# B&R Automation Studio project DuctLines (part 4)

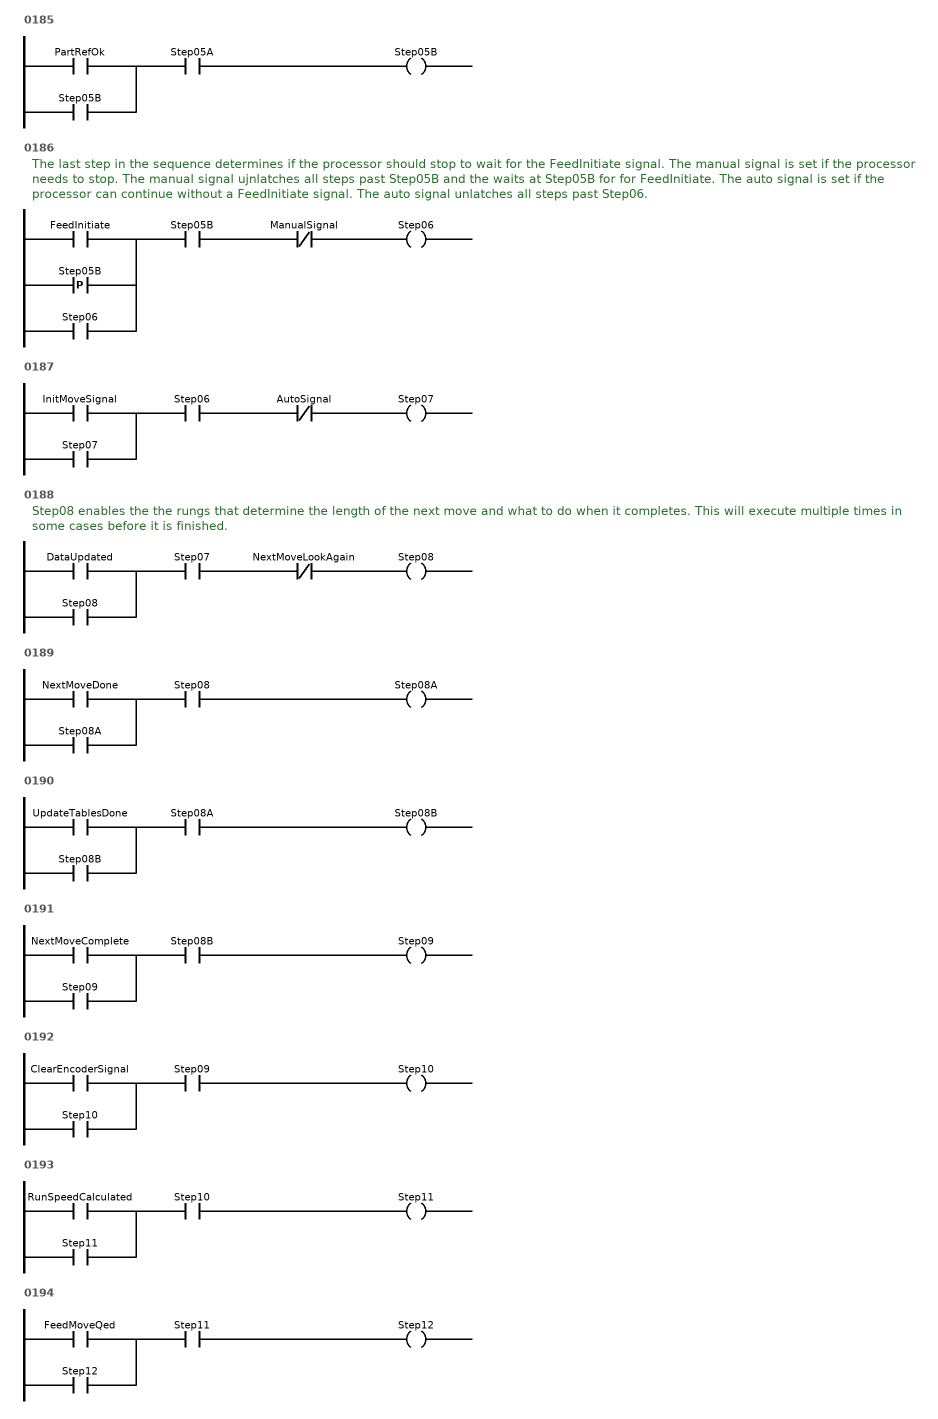
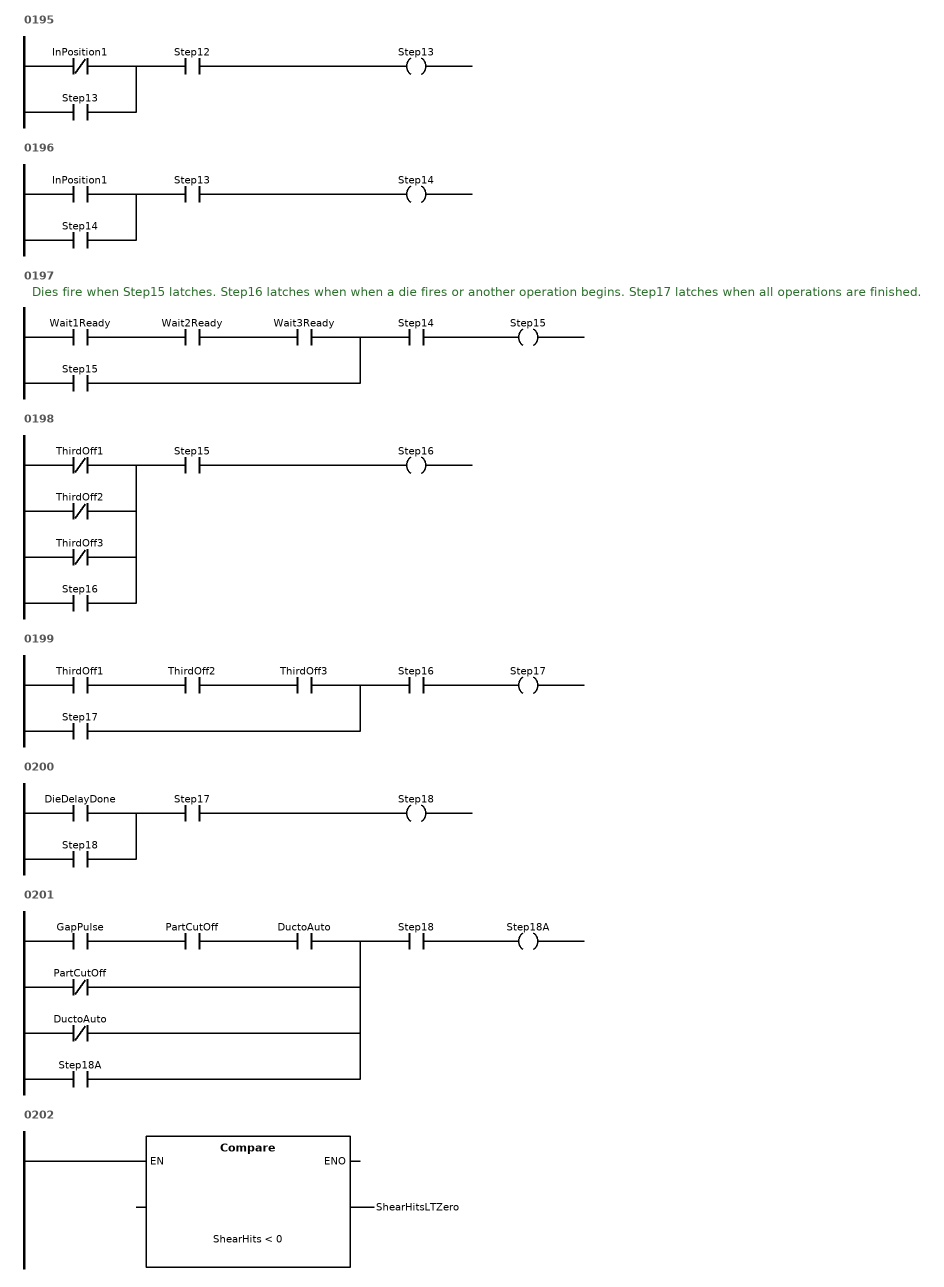
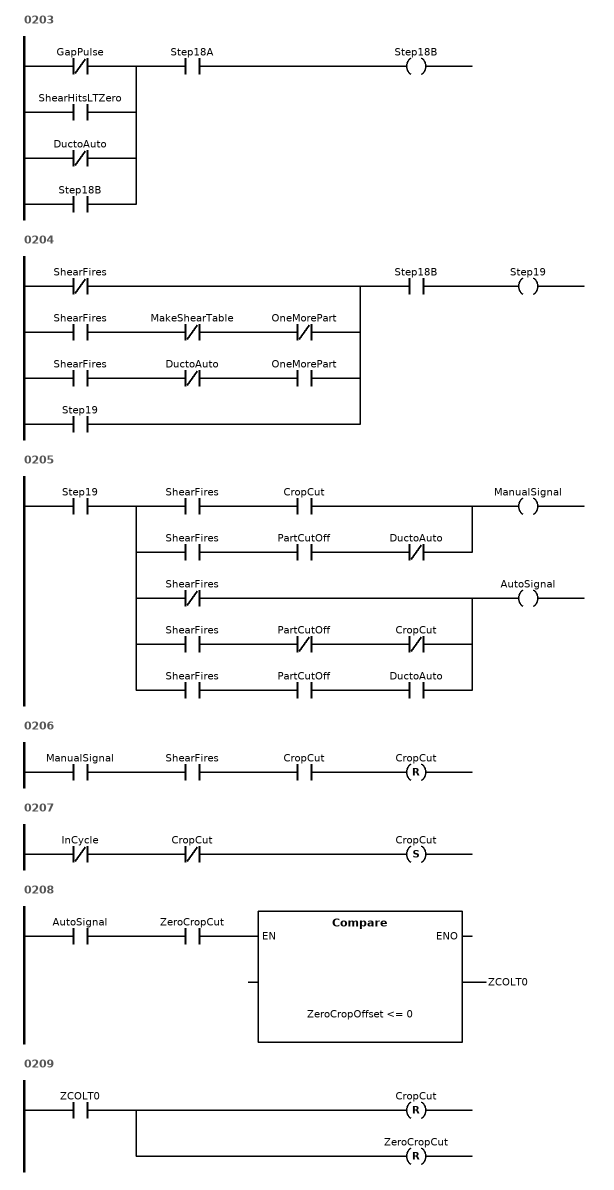
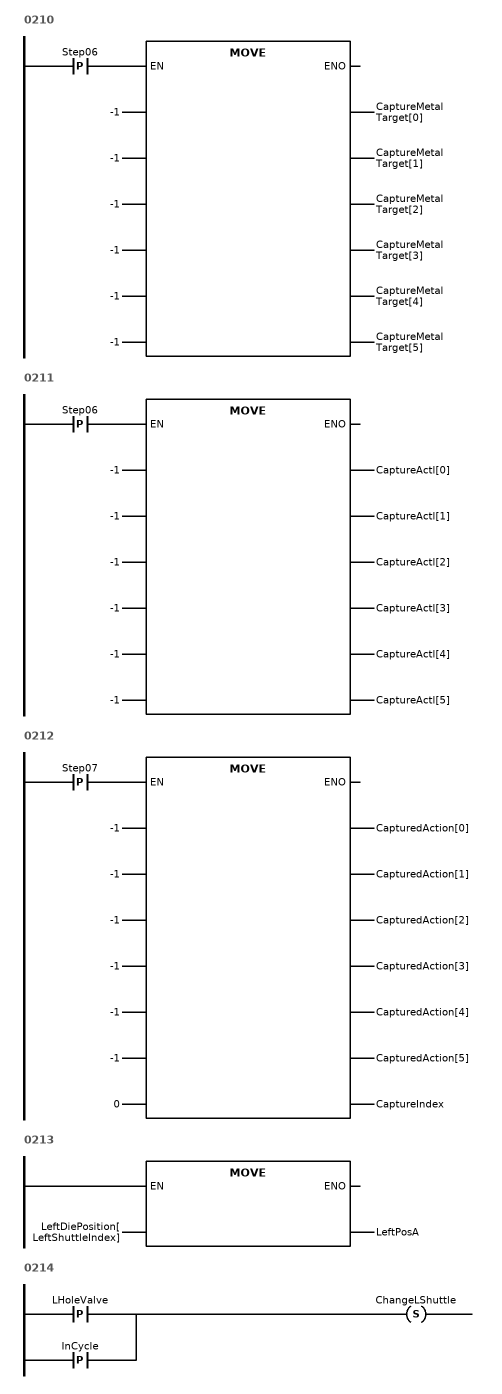
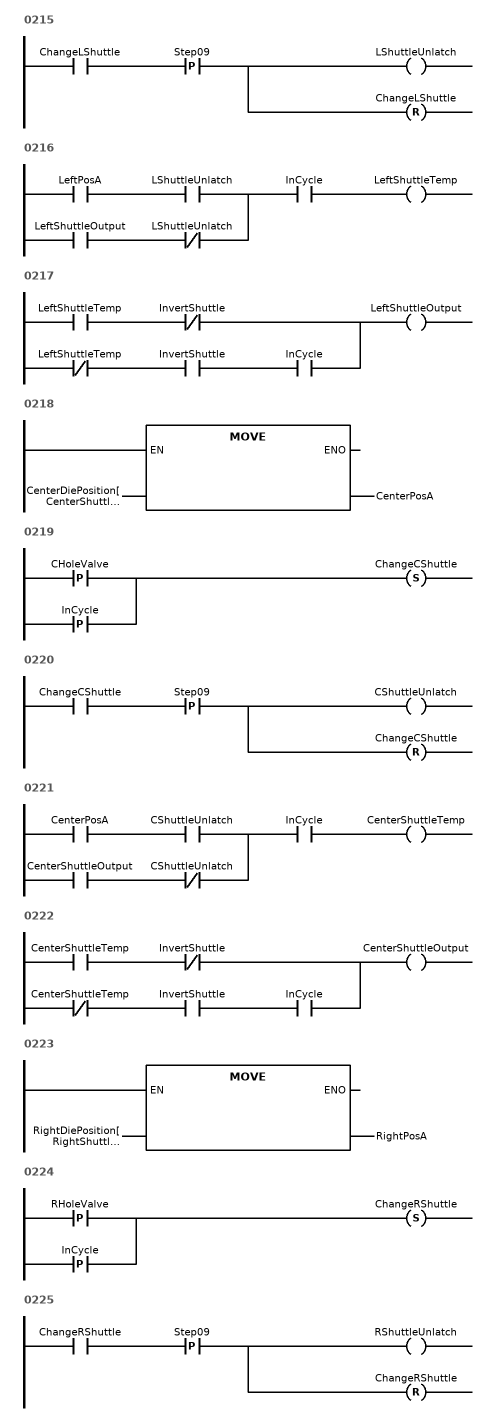
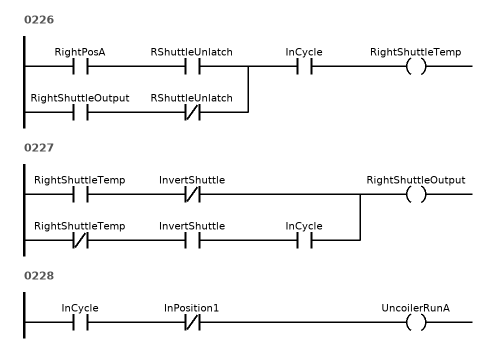
Ladder, written as Structured Text:
```iecst
PROGRAM _CYCLIC
VAR
    _e1 : R_TRIG;
    _e2 : R_TRIG;
    _e3 : F_TRIG;
    _e4 : F_TRIG;
    _e5 : R_TRIG;
    _e6 : F_TRIG;
    _e7 : F_TRIG;
    _e8 : F_TRIG;
    _e9 : R_TRIG;
    _p10 : BOOL;
    _e11 : R_TRIG;
    _e12 : R_TRIG;
    _e13 : R_TRIG;
    _e14 : F_TRIG;
    _e15 : F_TRIG;
    _e16 : R_TRIG;
    _e17 : R_TRIG;
    _e18 : R_TRIG;
    _e19 : R_TRIG;
    _e20 : R_TRIG;
    _e21 : R_TRIG;
    _e22 : R_TRIG;
    _e23 : R_TRIG;
    _e24 : R_TRIG;
    _e25 : R_TRIG;
    _e26 : R_TRIG;
    _e27 : R_TRIG;
    _e28 : F_TRIG;
    _e29 : R_TRIG;
    _e30 : R_TRIG;
    _e31 : F_TRIG;
    _e32 : R_TRIG;
    _e33 : R_TRIG;
    _e34 : R_TRIG;
    _e35 : R_TRIG;
    _e36 : F_TRIG;
    _e37 : R_TRIG;
    _e38 : F_TRIG;
    _e39 : R_TRIG;
    _e40 : F_TRIG;
    _e41 : R_TRIG;
    _e42 : F_TRIG;
    _e43 : R_TRIG;
    _e44 : F_TRIG;
    _e45 : R_TRIG;
    _e46 : F_TRIG;
    _e47 : R_TRIG;
    _e48 : F_TRIG;
    _e49 : R_TRIG;
    _e50 : F_TRIG;
    _e51 : R_TRIG;
    _e52 : F_TRIG;
    _e53 : R_TRIG;
    _e54 : F_TRIG;
    _e55 : R_TRIG;
    _e56 : F_TRIG;
    _e57 : R_TRIG;
    _e58 : R_TRIG;
    _e59 : R_TRIG;
    _e60 : R_TRIG;
    _e61 : R_TRIG;
    _e62 : R_TRIG;
    _e63 : R_TRIG;
    _e64 : R_TRIG;
    _e65 : R_TRIG;
    _e66 : R_TRIG;
    _e67 : R_TRIG;
    _e68 : R_TRIG;
    _e69 : R_TRIG;
    _e70 : R_TRIG;
    _e71 : R_TRIG;
    _e72 : R_TRIG;
    _e73 : R_TRIG;
    _e74 : R_TRIG;
    _e75 : F_TRIG;
    _e76 : R_TRIG;
    _e77 : R_TRIG;
    _e78 : R_TRIG;
    _e79 : R_TRIG;
    _e80 : R_TRIG;
    _e81 : R_TRIG;
    _e82 : R_TRIG;
    _e83 : F_TRIG;
    _e84 : R_TRIG;
    _e85 : R_TRIG;
    _e86 : R_TRIG;
    _e87 : R_TRIG;
    _e88 : R_TRIG;
    _e89 : R_TRIG;
    _p90 : BOOL;
    _e91 : F_TRIG;
    _e92 : R_TRIG;
    _e93 : R_TRIG;
    _e94 : R_TRIG;
    _e95 : R_TRIG;
    _e96 : R_TRIG;
    _e97 : R_TRIG;
    _e98 : R_TRIG;
    _e99 : R_TRIG;
    _e100 : R_TRIG;
    _e101 : R_TRIG;
    _e102 : R_TRIG;
    _e103 : R_TRIG;
    _e104 : R_TRIG;
    _e105 : R_TRIG;
END_VAR
(* Network 1 *)
MetalEncoder := ActlMetalEncoder - CoilAccumulator;

(* Network 2 *)
AmberLight := ProcessorDriveEnable;

(* Network 3 *)
Analog1Forward := (ProcessorDriveEnable AND ProcessorJogFwd AND NOT InCycle) OR (Step04C AND NOT Step04D);

(* Network 4 *)
Analog1Reverse := (ProcessorDriveEnable AND ProcessorJogRev AND NOT InCycle) OR (Step04 AND NOT Step04B);

(* Network 5 *)
_e1(CLK := Analog1Forward);
IF _e1.Q THEN MotionStatus1 := 4; END_IF;

(* Network 6 *)
_e2(CLK := Analog1Reverse);
IF _e2.Q THEN MotionStatus1 := 5; END_IF;

(* Network 7 *)
_e3(CLK := Analog1Forward);
_e4(CLK := Analog1Reverse);
IF (_e3.Q OR _e4.Q) AND NOT StopFlag1 THEN StopFlag1 := TRUE; END_IF;

(* Network 8: ElectricDriveEnable Output *)
ElectricDriveEnable := MotionStatus1 >= 0;

(* Network 9: Blocking Valve Output *)
BlockingValve := ElectricDriveEnable OR ForceBlockingValve;

(* Network 10 *)
_e5(CLK := Step04E);
IF _e5.Q THEN MotionStatus1 := 0; END_IF;

(* Network 11 *)
_e6(CLK := InCycle);
IF _e6.Q THEN MotionStatus1 := -1; END_IF;

(* Network 12 *)
_e7(CLK := ProcessorDriveEnable);
IF _e7.Q THEN MotionStatus1 := -1; END_IF;

(* Network 13 *)
ServoLoop1Closed := (MotionStatus1 >= 0) AND (MotionStatus1 <= 3);

(* Network 14 *)
_e8(CLK := HumpLimitSwitch);
IF _e8.Q AND ServoLoop1Closed THEN MotionStatus1 := -1; END_IF;

(* Network 15: OneMorePart logic needs To Execute Before The FeedInitiate Signal rung. *)
JobChanging := (RunJob - 1)  <> ShearJob;

(* Network 16 *)
OneMorePart := (InCycle OR (OneMorePart AND NOT FeedInitiate)) AND JobChanging AND NOT RunContinuousSignal;

(* Network 17: Feed Initiate Signal *)
_e9(CLK := FeedInitButton);
_p10 := _e9.Q AND ProcessorDriveEnable AND MatlAtMeasureRoll;
FeedInitiate := _p10 AND (NOT ShearBrakeInstalled OR ShearBrakeReady);

(* Network 18: Verify HMI Job change request *)
IF RunJobClick AND NOT InCycle THEN NewRunJobOk := NewRunJob <= MaxRunJob; END_IF;

(* Network 19 *)
IF RunJobClick AND NewRunJobOk AND NOT InCycle THEN RunJob := NewRunJob; END_IF;

(* Network 20 *)
IF RunJobClick THEN NewRunJobOk := FALSE; END_IF;

(* Network 21 *)
IF RunJobClick THEN RunJobClick := FALSE; END_IF;

(* Network 22: Update HMI job when the shear finishes one. *)
JobsDifferent := (RunJob - 1) <> ShearJob;

(* Network 23 *)
ChangeJob1 := InCycle AND Step19 AND ShearFires AND JobsDifferent;

(* Network 24 *)
IF ChangeJob1 THEN RunJob := ShearJob + 1; END_IF;

(* Network 25 *)
_e11(CLK := FeedInitiate);
IF _e11.Q THEN NoShearHits := FALSE; END_IF;

(* Network 26: Latch BatchActive in whenever the FeedInitiate signal comes on and the Ducto Sequence isn't started. Step04 latches after PC downloads tables and resets StartSignal. Unlatch BatchActive at that point if the shear has no hits. Step19 is the last one in the Ducto sequence. If there are no shear hits, the run is finished. BatchActive unlatches and the entire sequence unlatches. *)
_e12(CLK := Step04);
IF Step19 OR _e12.Q THEN NoShearHits := ShearHits < 0; END_IF;

(* Network 27 *)
_e13(CLK := WarningComplete);
_e14(CLK := HumpLimitSwitch);
_e15(CLK := MatlAtMeasureRoll);
BatchCancelUnlatch := BatchCancelSignal OR NoShearHits OR NOT ProcessorDriveEnable OR (_e13.Q AND NOT FeedInitButton) OR _e14.Q OR _e15.Q;

(* Network 28 *)
InCycle := ((FeedInitiate AND NOT Step01) OR InCycle) AND NOT BatchCancelUnlatch;

(* Network 29 *)
BlueLight := InCycle;

(* Network 30: Turn Off The BatchActivePhysical Output momentarily To Unlatch The Physical Auto Circuit *)
Block_1 := (Step18 AND OneMorePart) OR (Block_1 AND DuctoAuto);

(* Network 31 *)
BatchActivePhysical := InCycle AND NOT Block_1;

(* Network 32: There are 3 of these timers *)
ZRCTon(IN := Step04A AND NOT Step04B, PT := T#500ms);
ZCReverseComplete := ZRCTon.Q;

(* Network 33 *)
DDDoneTimer(IN := Step04B AND NOT Step04C, PT := T#2s);
DirectionDelayDone := DDDoneTimer.Q;

(* Network 34 *)
ZCSCTimer(IN := Step04D, PT := T#2s);
ZCSettleComplete := ZCSCTimer.Q;

(* Network 35 *)
_e16(CLK := MatlAtMeasureRoll);
IF _e16.Q AND Step04C AND NOT Step04D THEN MetalEncoderLatch := ActlMetalEncoder; END_IF;

(* Network 36 *)
_e17(CLK := Step05A);
IF _e17.Q AND NOT ZeroCropCut THEN MetalEncoderLatch := ActlMetalEncoder; END_IF;

(* Network 37: First actions in Ducto sequence, reset indexes and moves, set start signal for PC to generate die tables. *)
IF Step01 AND NOT Step02 THEN
    ShearMove := 0.0;
    LTNotchMove := 0.0;
    VNotchMove := 0.0;
    LeftHoleMove := 0.0;
    CenterHoleMove := 0.0;
    RightHoleMove := 0.0;
    PartsMade := 0;
    ShearIndex := 0;
    LTNotchIndex := 0;
    VNotchIndex := 0;
    LeftHoleIndex := 0;
    CenterHoleIndex := 0;
    RightHoleIndex := 0;
    ButtonMove := 0.0;
    ShearBrakeMove := 0.0;
    CustomLTMove := 0.0;
    CleatMove := 0.0;
    ButtonIndex := 0;
    ShearBrakeIndex := 0;
    CustomLTIndex := 0;
END_IF;

(* Network 38 *)
IF Step01 AND NOT Step02 THEN
    CleatIndex := 0;
    ButtonActual := 0;
    CustomVMove := 0.0;
    CustomVIndex := 0;
    BeadRollMove := 0.0;
    BeadRollIndex := 0;
    StartSignal := TRUE;
END_IF;

(* Network 39 *)
TON_2(IN := Step02 AND NOT Step03, PT := WarningDelay1);
WarningComplete := TON_2.Q;

(* Network 40 *)
WarningHorn := Step02 AND NOT Step03;

(* Network 41: The Actual Material Counter Needs To Be Initialized To ZeroCropDifference Here, too. *)
_e18(CLK := Step05A);
IF _e18.Q THEN
    ZeroCropDifference := MetalEncoderLatch - ActlMetalEncoder;
    CoilAccumulator := ZeroCropDifference;
    MetalTarget := ZeroCropDifference;
END_IF;

(* Network 42 *)
TON_1(IN := Step05A, PT := T#200ms);
PartRefOk := TON_1.Q;

(* Network 43 *)
ProcessorEncoderReset := (Step05A AND NOT Step05B) OR (ShearValve AND NOT InCycle);

(* Network 44: Reset variable to get ready for a new move *)
IF Step06 AND NOT Step07 THEN
    PartCutOff := FALSE;
    ShearFires := FALSE;
    IncrementalRealTarget := 0.0;
END_IF;
InitMoveSignal := Step06 AND NOT Step07;

(* Network 45: Make Sure All Data Is Updated By PC *)
HalfUpdated1 := NOT MakeShearTable AND NOT MakeLTTable AND NOT MakeVTable AND NOT MakeLHoleTable AND NOT MakeCHoleTable AND NOT MakeBeadRollTable;

(* Network 46 *)
HalfUpdated2 := NOT MakeRHoleTable AND NOT MakeButtonTable AND NOT MakeShearBrakeTable AND NOT MakeCustomLTTable AND NOT MakeCleatTable AND NOT MakeCustomVTable;

(* Network 47 *)
DataUpdated := HalfUpdated1 AND HalfUpdated2;

(* Network 48: New Connector Logic *)
_e19(CLK := Step04);
IF _e19.Q THEN SavedConnector := LatestConnector; END_IF;

(* Network 49 *)
_e20(CLK := Step08);
IF _e20.Q THEN SetConnectorChange := (LatestConnector <> SavedConnector) AND (LTNotchHits > 0); END_IF;

(* Network 50 *)
ChangeConnector := SetConnectorChange OR (ChangeConnector AND NOT LTValve AND InCycle);

(* Network 51: Net #37-40 from PicPro.  *)
MUX1:
_e21(CLK := Step08);
IF _e21.Q AND ShearUsedUp THEN
    ShearMove := MUX(K := ShearIndex, IN2 := ShearTable[0], IN3 := ShearTable[1], IN4 := ShearTable[2], IN5 := ShearTable[3], IN6 := ShearTable[4], IN7 := ShearTable[5]);
END_IF;
IF _e21.Q AND LTUsedUp THEN
    LTNotchMove := MUX(K := LTNotchIndex, IN2 := LTNotchTable[0], IN3 := LTNotchTable[1], IN4 := LTNotchTable[2], IN5 := LTNotchTable[3], IN6 := LTNotchTable[4], IN7 := LTNotchTable[5]);
END_IF;
IF _e21.Q AND VUsedUp THEN
    VNotchMove := MUX(K := VNotchIndex, IN2 := VNotchTable[0], IN3 := VNotchTable[1], IN4 := VNotchTable[2], IN5 := VNotchTable[3], IN6 := VNotchTable[4], IN7 := VNotchTable[5]);
END_IF;

(* Network 52 *)
_e22(CLK := Step08);
IF _e22.Q AND ButtonUsedUp THEN
    ButtonMove := MUX(K := ButtonIndex, IN2 := ButtonTable[0], IN3 := ButtonTable[1], IN4 := ButtonTable[2], IN5 := ButtonTable[3], IN6 := ButtonTable[4], IN7 := ButtonTable[5]);
END_IF;
IF _e22.Q AND ShearBrakeUsedUp THEN
    ShearBrakeMove := MUX(K := ShearBrakeIndex, IN2 := ShearBrakeTable[0], IN3 := ShearBrakeTable[1], IN4 := ShearBrakeTable[2], IN5 := ShearBrakeTable[3], IN6 := ShearBrakeTable[4], IN7 := ShearBrakeTable[5]);
END_IF;
IF _e22.Q AND CustomLTUsedUp THEN
    CustomLTMove := MUX(K := CustomLTIndex, IN2 := CustomLTTable[0], IN3 := CustomLTTable[1], IN4 := CustomLTTable[2], IN5 := CustomLTTable[3], IN6 := CustomLTTable[4], IN7 := CustomLTTable[5]);
END_IF;

(* Network 53 *)
_e23(CLK := Step08);
IF _e23.Q AND CleatUsedUp THEN
    CleatMove := MUX(K := CleatIndex, IN2 := CleatTable[0], IN3 := CleatTable[1], IN4 := CleatTable[2], IN5 := CleatTable[3], IN6 := CleatTable[4], IN7 := CleatTable[5]);
END_IF;
IF _e23.Q AND CustomVUsedUp THEN
    CustomVMove := MUX(K := CustomVIndex, IN2 := CustomVTable[0], IN3 := CustomVTable[1], IN4 := CustomVTable[2], IN5 := CustomVTable[3], IN6 := CustomVTable[4], IN7 := CustomVTable[5]);
END_IF;

(* Network 54: These 4 tables have too many values for the B&R mux. *)
_e24(CLK := Step08);
IF _e24.Q AND LeftHoleUsedUp THEN LeftHoleMove := LeftHoleTable[LeftHoleIndex]; END_IF;
IF _e24.Q AND CenterHoleUsedUp THEN CenterHoleMove := CenterHoleTable[CenterHoleIndex]; END_IF;
IF _e24.Q AND RightHoleUsedUp THEN RightHoleMove := RightHoleTable[RightHoleIndex]; END_IF;
IF _e24.Q AND BeadRollUsedUp THEN BeadRollMove := BeadRollTable[BeadRollIndex]; END_IF;

(* Network 55 *)
_e25(CLK := Step08);
IF _e25.Q THEN
    LeftShuttleIndex := LeftHoleIndex;
    CenterShuttleIndex := CenterHoleIndex;
    RightShuttleIndex := RightHoleIndex;
END_IF;

(* Network 56 *)
_e26(CLK := Step08);
IF _e26.Q THEN getNextMove; END_IF;

(* Network 57 *)
_e27(CLK := Step08A);
_e28(CLK := InCycle);
IF _e27.Q OR _e28.Q THEN NextMoveDone := FALSE; END_IF;

(* Network 58 *)
ShearUsedUp := ABS(ShearMove) <= InPositionBand;

(* Network 59 *)
LTUsedUp := ABS(LTNotchMove) <= InPositionBand;

(* Network 60 *)
VUsedUp := ABS(VNotchMove) <= InPositionBand;

(* Network 61 *)
LeftHoleUsedUp := ABS(LeftHoleMove) <= InPositionBand;

(* Network 62 *)
CenterHoleUsedUp := ABS(CenterHoleMove) <= InPositionBand;

(* Network 63 *)
RightHoleUsedUp := ABS(RightHoleMove) <= InPositionBand;

(* Network 64 *)
ButtonUsedUp := ABS(ButtonMove) <= InPositionBand;

(* Network 65 *)
ShearBrakeUsedUp := ABS(ShearBrakeMove) <= InPositionBand;

(* Network 66 *)
CustomLTUsedUp := ABS(CustomLTMove) <= InPositionBand;

(* Network 67 *)
CleatUsedUp := ABS(CleatMove) <= InPositionBand;

(* Network 68 *)
CustomVUsedUp := ABS(CustomVMove) <= InPositionBand;

(* Network 69 *)
BeadRollUsedUp := ABS(BeadRollMove) <= InPositionBand;

(* Network 70 *)
_e29(CLK := Step08A);
IF _e29.Q THEN UpdateTables; END_IF;

(* Network 71 *)
_e30(CLK := Step08B);
_e31(CLK := InCycle);
IF _e30.Q OR _e31.Q THEN UpdateTablesDone := FALSE; END_IF;

(* Network 72 *)
_e32(CLK := Step08B);
IF _e32.Q THEN IncrementalRealTarget := IncrementalRealTarget + SmallResult; END_IF;

(* Network 73 *)
_e33(CLK := Step08B);
NextMoveComplete := _e33.Q AND (ShearFires OR LTFires OR VFires OR LeftHoleFires OR CenterHoleFires OR RightHoleFires OR ButtonFires OR ShearBrakeFires OR CustomLTFires OR CleatFires OR CustomVFires OR BeadRollFires);

(* Network 74 *)
_e34(CLK := Step08B);
NextMoveLookAgain := _e34.Q AND NOT NextMoveComplete;

(* Network 75 *)
_e35(CLK := LTValve);
_e36(CLK := InCycle);
IF _e35.Q OR _e36.Q THEN LTFires := FALSE; END_IF;

(* Network 76 *)
_e37(CLK := VValve);
_e38(CLK := InCycle);
IF _e37.Q OR _e38.Q THEN VFires := FALSE; END_IF;

(* Network 77 *)
_e39(CLK := LHoleValve);
_e40(CLK := InCycle);
IF _e39.Q OR _e40.Q THEN LeftHoleFires := FALSE; END_IF;

(* Network 78 *)
_e41(CLK := CHoleValve);
_e42(CLK := InCycle);
IF _e41.Q OR _e42.Q THEN CenterHoleFires := FALSE; END_IF;

(* Network 79 *)
_e43(CLK := RHoleValve);
_e44(CLK := InCycle);
IF _e43.Q OR _e44.Q THEN RightHoleFires := FALSE; END_IF;

(* Network 80 *)
_e45(CLK := CycleButtons);
_e46(CLK := InCycle);
IF _e45.Q OR _e46.Q THEN ButtonFires := FALSE; END_IF;

(* Network 81 *)
_e47(CLK := CycleMaleBender);
_e48(CLK := InCycle);
IF _e47.Q OR _e48.Q THEN ShearBrakeFires := FALSE; END_IF;

(* Network 82 *)
_e49(CLK := CustomLTValve);
_e50(CLK := InCycle);
IF _e49.Q OR _e50.Q THEN CustomLTFires := FALSE; END_IF;

(* Network 83 *)
_e51(CLK := ChangeKDRolls);
_e52(CLK := InCycle);
IF _e51.Q OR _e52.Q THEN CleatFires := FALSE; END_IF;

(* Network 84 *)
_e53(CLK := CustomVValve);
_e54(CLK := InCycle);
IF _e53.Q OR _e54.Q THEN CustomVFires := FALSE; END_IF;

(* Network 85 *)
_e55(CLK := WaitCon3);
_e56(CLK := InCycle);
IF _e55.Q OR _e56.Q THEN BeadRollFires := FALSE; END_IF;

(* Network 86 *)
_e57(CLK := Step09);
IF _e57.Q THEN MetalScaler := MetalDesired / MetalActual; END_IF;
ClearEncoderSignal := _e57.Q;

(* Network 87 *)
_e58(CLK := Step10);
IF _e58.Q AND CropCut THEN RunSpeed1 := CropPercent1; END_IF;
IF _e58.Q AND NOT CropCut THEN RunSpeed1 := PercentSpeed1; END_IF;
RunSpeedCalculated := _e58.Q;

(* Network 88 *)
IF Step11 AND NOT Step12 THEN MotionStatus1 := 1; END_IF;
FeedMoveQed := Step11 AND NOT Step12;

(* Network 89 *)
WaitToFire1 := Step14 AND LTFires AND ChangeConnector;
WaitCon1 := Step14 AND FeedInitiate;

(* Network 90 *)
TON_10(IN := WaitToFire2, PT := T#50ms);
WaitCon2 := TON_10.Q;

(* Network 91 *)
_e59(CLK := InPosition1);
WaitToFire2 := (_e59.Q OR WaitToFire2) AND NOT WaitCon2;

(* Network 92 *)
WaitCon3 := Step14 AND BeadRollFires AND FeedInitiate;
WaitToFire3 := Step14 AND BeadRollFires;

(* Network 93 *)
_e60(CLK := WaitToFire3);
IF _e60.Q THEN ChangeBeadRoll := TRUE; END_IF;

(* Network 94 *)
Wait1Ready := Step14 AND ((WaitToFire1 AND WaitCon1) OR NOT WaitToFire1);
Wait2Ready := Step14 AND ((WaitToFire2 AND WaitCon2) OR NOT WaitToFire2);
Wait3Ready := Step14 AND ((WaitToFire3 AND WaitCon3) OR NOT WaitToFire3);

(* Network 95 *)
_e61(CLK := Step15);
IF _e61.Q THEN
    CaptureMetalTarget[CaptureIndex] := MetalTarget;
    CaptureActl[CaptureIndex] := ActlMetalEncoder;
END_IF;

(* Network 96 *)
_e62(CLK := Step15);
IF _e62.Q AND ShearFires THEN CapturedAction[CaptureIndex] := 1; END_IF;

(* Network 97 *)
_e63(CLK := Step15);
IF _e63.Q AND LTFires THEN CapturedAction[CaptureIndex] := 2; END_IF;

(* Network 98 *)
_e64(CLK := Step15);
IF _e64.Q AND VFires THEN CapturedAction[CaptureIndex] := 3; END_IF;

(* Network 99 *)
_e65(CLK := Step15);
IF _e65.Q THEN CaptureIndex := CaptureIndex + 1; END_IF;

(* Network 100 *)
ShearTemp := (Step15 AND ShearFires) OR (NOT InCycle AND CycleShear);

(* Network 101 *)
IF CycleShear THEN CycleShear := FALSE; END_IF;

(* Network 102 *)
_e66(CLK := ShearTemp);
IF _e66.Q THEN shearTime := DINT_TO_TIME(ShearDwell); END_IF;

(* Network 103 *)
TP_0(IN := ShearTemp, PT := shearTime);
ShearValve := TP_0.Q;

(* Network 104 *)
LTTemp := (Step15 AND LTFires) OR (NOT InCycle AND CycleLTDie);

(* Network 105 *)
IF CycleLTDie THEN CycleLTDie := FALSE; END_IF;

(* Network 106 *)
_e67(CLK := LTTemp);
IF _e67.Q THEN LTTime := DINT_TO_TIME(LTDwell); END_IF;

(* Network 107 *)
TP_1(IN := LTTemp, PT := LTTime);
LTValve := TP_1.Q;

(* Network 108 *)
VTemp := (Step15 AND VFires) OR (NOT InCycle AND CycleVDie);

(* Network 109 *)
IF CycleVDie THEN CycleVDie := FALSE; END_IF;

(* Network 110 *)
_e68(CLK := VTemp);
IF _e68.Q THEN VTime := DINT_TO_TIME(VDwell); END_IF;

(* Network 111 *)
TP_2(IN := VTemp, PT := VTime);
VValve := TP_2.Q;

(* Network 112 *)
LHTemp := (Step15 AND LeftHoleFires) OR (NOT InCycle AND CycleLDie);

(* Network 113 *)
IF CycleLDie THEN CycleLDie := FALSE; END_IF;

(* Network 114 *)
_e69(CLK := LHTemp);
IF _e69.Q THEN LeftHoleTime := DINT_TO_TIME(LHoleDwell); END_IF;

(* Network 115 *)
TP_3(IN := LHTemp, PT := LeftHoleTime);
LHoleValve := TP_3.Q;

(* Network 116 *)
CHTemp := (Step15 AND CenterHoleFires) OR (NOT InCycle AND CycleCDie);

(* Network 117 *)
IF CycleCDie THEN CycleCDie := FALSE; END_IF;

(* Network 118 *)
_e70(CLK := CHTemp);
IF _e70.Q THEN CenterHoleTime := DINT_TO_TIME(CHoleDwell); END_IF;

(* Network 119 *)
TP_4(IN := CHTemp, PT := CenterHoleTime);
CHoleValve := TP_4.Q;

(* Network 120 *)
RHTemp := (Step15 AND RightHoleFires) OR (NOT InCycle AND CycleRDie);

(* Network 121 *)
IF CycleRDie THEN CycleRDie := FALSE; END_IF;

(* Network 122 *)
_e71(CLK := RHTemp);
IF _e71.Q THEN RightHoleTime := DINT_TO_TIME(RHoleDwell); END_IF;

(* Network 123 *)
TP_5(IN := RHTemp, PT := RightHoleTime);
RHoleValve := TP_5.Q;

(* Network 124 *)
CLTTemp := (Step15 AND CustomLTFires) OR (NOT InCycle AND CycleCustomLTDie);

(* Network 125 *)
IF CycleCustomLTDie THEN CycleCustomLTDie := FALSE; END_IF;

(* Network 126 *)
_e72(CLK := CLTTemp);
IF _e72.Q THEN CustomLTTime := DINT_TO_TIME(CustomLTDwell); END_IF;

(* Network 127 *)
TP_6(IN := CLTTemp, PT := CustomLTTime);
CustomLTValve := TP_6.Q;

(* Network 128 *)
CustomVTemp := (Step15 AND CustomVFires) OR (NOT InCycle AND CycleCustomVDie);

(* Network 129 *)
IF CycleCustomVDie THEN CycleCustomVDie := FALSE; END_IF;

(* Network 130 *)
_e73(CLK := CustomVTemp);
IF _e73.Q THEN CustomVTime := DINT_TO_TIME(CustomVDwell); END_IF;

(* Network 131 *)
TP_7(IN := CustomVTemp, PT := CustomVTime);
CustomVValve := TP_7.Q;

(* Network 132 *)
OneInchHolePunch := CustomVValve;

(* Network 133 *)
_e74(CLK := ButtonBack7);
_e75(CLK := InCycle);
UnlatchButtons := (Step15 AND _e74.Q) OR _e75.Q;

(* Network 134 *)
_e76(CLK := Step15);
CycleButtons := ((_e76.Q AND ButtonFires) OR CycleButtons) AND NOT UnlatchButtons;

(* Network 135: Convert Presets And Turn Button Gag On, Start Clamp Delay Timer. *)
_e77(CLK := CycleButtons);
SnapButton1 := (_e77.Q OR SnapButton1) AND InCycle AND NOT SnapButton7;

(* Network 136: Turn Shear Brake Clamp On, Start Dwell Timer *)
SnapButton2 := (TON_3Done OR SnapButton2) AND SnapButton1;

(* Network 137: Turn Shear Brake Clamp Off, Start Timer *)
SnapButton3 := (TON_4Done OR SnapButton3) AND SnapButton2;

(* Network 138 *)
SnapButton3A := (ShearClampUpProx OR SnapButton3A) AND SnapButton3;

(* Network 139: Turn Button Gag Off,Do Nothing For 250 ms. *)
SnapButton4 := (TON_5Done OR SnapButton4) AND SnapButton3;

(* Network 140: Back Material Up 1/16" And Wait 500 ms. For It. *)
SnapButton5 := (TON_6Done OR SnapButton5) AND SnapButton4;

(* Network 141: Snap Lock Sequence Complete *)
SnapButton6 := (TON_7Done OR SnapButton6) AND SnapButton5;

(* Network 142 *)
SnapButton7 := (TON_8Done OR SnapButton7) AND SnapButton6;

(* Network 143 *)
ButtonBack7 := SnapButton7;

(* Network 144 *)
_e78(CLK := SnapButton1);
IF _e78.Q THEN SBClampDelay := DINT_TO_TIME(BDelay1); END_IF;

(* Network 145 *)
_e79(CLK := SnapButton1);
IF _e79.Q THEN SBClampDwell := DINT_TO_TIME(BDelay2); END_IF;

(* Network 146 *)
TON_3(IN := SnapButton1, PT := SBClampDelay);
TON_3Done := TON_3.Q;

(* Network 147 *)
TON_4(IN := SnapButton2, PT := SBClampDwell);
TON_4Done := TON_4.Q;

(* Network 148 *)
TON_5(IN := SnapButton3, PT := SBClampDelay);
TON_5Done := TON_5.Q;

(* Network 149 *)
TON_6(IN := SnapButton4, PT := T#300ms);
TON_6Done := TON_6.Q;

(* Network 150: Change Metal Target. Motion Control hold routine should respond to this small change. *)
_e80(CLK := SnapButton5);
IF _e80.Q THEN MetalTarget := MetalTarget - REAL_TO_DINT(UnitsPerInch1/8.0); END_IF;

(* Network 151: Change Metal Target Back. Motion Control hold routine should respond to this small change. *)
_e81(CLK := SnapButton6);
IF _e81.Q THEN MetalTarget := MetalTarget + REAL_TO_DINT(UnitsPerInch1/8.0); END_IF;

(* Network 152 *)
TON_7(IN := SnapButton5, PT := T#10ms);
TON_7Done := TON_7.Q;

(* Network 153 *)
TON_8(IN := SnapButton6, PT := T#100ms);
TON_8Done := TON_8.Q;

(* Network 154 *)
SnapLockButtonGag := SnapButton1 AND NOT SnapButton3A;

(* Network 155 *)
ShearClamp4Buttons := SnapButton2 AND NOT SnapButton3;

(* Network 156 *)
_e82(CLK := ShearClampUpProx);
_e83(CLK := ProcessorDriveEnable);
UnlatchBender := ((Step15 OR ShearBrakeLatch) AND _e82.Q) OR _e83.Q;

(* Network 157 *)
IF UnlatchBender THEN ShearBrakeLatch := FALSE; END_IF;

(* Network 158 *)
_e84(CLK := Step15);
CycleMaleBender := ((_e84.Q AND ShearBrakeFires) OR ShearBrakeLatch OR CycleMaleBender) AND NOT UnlatchBender;

(* Network 159 *)
_e85(CLK := Step15);
ChangeKDRolls := _e85.Q AND CleatFires;

(* Network 160 *)
LeftKnockDownRoll := (ChangeKDRolls AND LeftCleatEnable AND NOT LeftKnockDownRoll) OR (LeftKnockDownRoll AND InCycle AND NOT ChangeKDRolls);

(* Network 161 *)
RightKnockDownRoll := (ChangeKDRolls AND RightCleatEnable AND NOT RightKnockDownRoll) OR (RightKnockDownRoll AND InCycle AND NOT ChangeKDRolls);

(* Network 162 *)
ThirdOff1 := NOT ShearValve AND NOT LTValve AND NOT VValve AND NOT LHoleValve;

(* Network 163 *)
ThirdOff2 := NOT CHoleValve AND NOT RHoleValve AND NOT ChangeKDRolls AND NOT CycleMaleBender;

(* Network 164 *)
ThirdOff3 := NOT CycleButtons AND NOT CustomLTValve AND NOT CustomVValve AND NOT WaitCon3;

(* Network 165 *)
_e86(CLK := Step17);
IF _e86.Q THEN DieUpTime := DINT_TO_TIME(DieUpDelay); END_IF;

(* Network 166 *)
TON_0(IN := Step17 AND NOT Step18, PT := DieUpTime);
DieDelayDone := TON_0.Q;

(* Network 167 *)
IncPartsMade := PartCutOff;

(* Network 168 *)
_e87(CLK := Step18);
IF _e87.Q THEN GTime := DINT_TO_TIME(GapTime); END_IF;

(* Network 169 *)
TP_8(IN := Step18 AND PartCutOff AND DuctoAuto, PT := GTime);
GapTP := TP_8.Q;

(* Network 170 *)
_e88(CLK := Step18);
GapPulse := GapTP OR _e88.Q;

(* Network 171 *)
_e89(CLK := Step18);
IF _e89.Q AND IncPartsMade THEN
    PartsMade := PartsMade + 1;
    RTotalInches := PartLength + RTotalInches;
    MarkAccumulator := PartLength + MarkAccumulator;
END_IF;

(* Network 172 *)
IF ChangeJob1 THEN PartsMade := 0; END_IF;

(* Network 173 *)
TotalInches := RTotalInches;

(* Network 174 *)
IF ClearLengthCountSignal THEN RTotalInches := 0; END_IF;
_p90 := ClearLengthCountSignal;
IF _p90 THEN ClearLengthCountSignal := FALSE; END_IF;

(* Network 175: Set StartSignal for touchscreen. Do the warning while waiting for data. Touchscreen resets StartSignal at the tail end of the data transfer. *)
Step01 := (FeedInitiate OR Step01) AND InCycle;

(* Network 176 *)
Step02 := (StartSignal OR Step02) AND Step01;

(* Network 177 *)
Step03 := (WarningComplete OR Step03) AND Step02;

(* Network 178 *)
Step04 := (NOT StartSignal OR Step04) AND Step03;

(* Network 179: Position material for no crop cut. Latch these rungs in if crop cutting. *)
_e91(CLK := MatlAtMeasureRoll);
Step04A := (_e91.Q OR NOT ZeroCropCut OR Step04A) AND Step04;

(* Network 180 *)
Step04B := (ZCReverseComplete OR NOT ZeroCropCut OR Step04B) AND Step04A;

(* Network 181 *)
Step04C := (DirectionDelayDone OR NOT ZeroCropCut OR Step04C) AND Step04B;

(* Network 182 *)
_e92(CLK := MatlAtMeasureRoll);
Step04D := (_e92.Q OR NOT ZeroCropCut OR Step04D) AND Step04C;

(* Network 183 *)
Step04E := (ZCSettleComplete OR NOT ZeroCropCut OR Step04E) AND Step04D;

(* Network 184 *)
Step05A := (ServoLoop1Closed OR Step05A) AND Step04E;

(* Network 185 *)
Step05B := (PartRefOk OR Step05B) AND Step05A;

(* Network 186: The last step in the sequence determines if the processor should stop to wait for the FeedInitiate signal. The manual signal is set if the processor needs to stop. The manual signal ujnlatches all steps past Step05B and the waits at Step05B for for FeedInitiate. The auto signal is set if the processor can continue without a FeedInitiate signal. The auto signal unlatches all steps past Step06. *)
_e93(CLK := Step05B);
Step06 := (FeedInitiate OR _e93.Q OR Step06) AND Step05B AND NOT ManualSignal;

(* Network 187 *)
Step07 := (InitMoveSignal OR Step07) AND Step06 AND NOT AutoSignal;

(* Network 188: Step08 enables the the rungs that determine the length of the next move and what to do when it completes. This will execute multiple times in some cases before it is finished. *)
Step08 := (DataUpdated OR Step08) AND Step07 AND NOT NextMoveLookAgain;

(* Network 189 *)
Step08A := (NextMoveDone OR Step08A) AND Step08;

(* Network 190 *)
Step08B := (UpdateTablesDone OR Step08B) AND Step08A;

(* Network 191 *)
Step09 := (NextMoveComplete OR Step09) AND Step08B;

(* Network 192 *)
Step10 := (ClearEncoderSignal OR Step10) AND Step09;

(* Network 193 *)
Step11 := (RunSpeedCalculated OR Step11) AND Step10;

(* Network 194 *)
Step12 := (FeedMoveQed OR Step12) AND Step11;

(* Network 195 *)
Step13 := (NOT InPosition1 OR Step13) AND Step12;

(* Network 196 *)
Step14 := (InPosition1 OR Step14) AND Step13;

(* Network 197: Dies fire when Step15 latches. Step16 latches when when a die fires or another operation begins. Step17 latches when all operations are finished. *)
Step15 := ((Wait1Ready AND Wait2Ready AND Wait3Ready) OR Step15) AND Step14;

(* Network 198 *)
Step16 := (NOT ThirdOff1 OR NOT ThirdOff2 OR NOT ThirdOff3 OR Step16) AND Step15;

(* Network 199 *)
Step17 := ((ThirdOff1 AND ThirdOff2 AND ThirdOff3) OR Step17) AND Step16;

(* Network 200 *)
Step18 := (DieDelayDone OR Step18) AND Step17;

(* Network 201 *)
Step18A := ((GapPulse AND PartCutOff AND DuctoAuto) OR NOT PartCutOff OR NOT DuctoAuto OR Step18A) AND Step18;

(* Network 202 *)
ShearHitsLTZero := ShearHits < 0;

(* Network 203 *)
Step18B := (NOT GapPulse OR ShearHitsLTZero OR NOT DuctoAuto OR Step18B) AND Step18A;

(* Network 204 *)
Step19 := (NOT ShearFires OR (ShearFires AND ((NOT MakeShearTable AND NOT OneMorePart) OR (NOT DuctoAuto AND OneMorePart))) OR Step19) AND Step18B;

(* Network 205 *)
ManualSignal := Step19 AND ShearFires AND (CropCut OR (PartCutOff AND NOT DuctoAuto));
AutoSignal := Step19 AND (NOT ShearFires OR (ShearFires AND ((NOT PartCutOff AND NOT CropCut) OR (PartCutOff AND DuctoAuto))));

(* Network 206 *)
IF ManualSignal AND ShearFires AND CropCut THEN CropCut := FALSE; END_IF;

(* Network 207 *)
IF NOT InCycle AND NOT CropCut THEN CropCut := TRUE; END_IF;

(* Network 208 *)
IF AutoSignal AND ZeroCropCut THEN ZCOLT0 := ZeroCropOffset <= 0; END_IF;

(* Network 209 *)
IF ZCOLT0 THEN
    CropCut := FALSE;
    ZeroCropCut := FALSE;
END_IF;

(* Network 210 *)
_e94(CLK := Step06);
IF _e94.Q THEN
    CaptureMetalTarget[0] := -1;
    CaptureMetalTarget[1] := -1;
    CaptureMetalTarget[2] := -1;
    CaptureMetalTarget[3] := -1;
    CaptureMetalTarget[4] := -1;
    CaptureMetalTarget[5] := -1;
END_IF;

(* Network 211 *)
_e95(CLK := Step06);
IF _e95.Q THEN
    CaptureActl[0] := -1;
    CaptureActl[1] := -1;
    CaptureActl[2] := -1;
    CaptureActl[3] := -1;
    CaptureActl[4] := -1;
    CaptureActl[5] := -1;
END_IF;

(* Network 212 *)
_e96(CLK := Step07);
IF _e96.Q THEN
    CapturedAction[0] := -1;
    CapturedAction[1] := -1;
    CapturedAction[2] := -1;
    CapturedAction[3] := -1;
    CapturedAction[4] := -1;
    CapturedAction[5] := -1;
    CaptureIndex := 0;
END_IF;

(* Network 213 *)
LeftPosA := LeftDiePosition[LeftShuttleIndex];

(* Network 214 *)
_e97(CLK := LHoleValve);
_e98(CLK := InCycle);
IF _e97.Q OR _e98.Q THEN ChangeLShuttle := TRUE; END_IF;

(* Network 215 *)
_e99(CLK := Step09);
LShuttleUnlatch := ChangeLShuttle AND _e99.Q;
IF ChangeLShuttle AND _e99.Q THEN ChangeLShuttle := FALSE; END_IF;

(* Network 216 *)
LeftShuttleTemp := ((LeftPosA AND LShuttleUnlatch) OR (LeftShuttleOutput AND NOT LShuttleUnlatch)) AND InCycle;

(* Network 217 *)
LeftShuttleOutput := (LeftShuttleTemp AND NOT InvertShuttle) OR (NOT LeftShuttleTemp AND InvertShuttle AND InCycle);

(* Network 218 *)
CenterPosA := CenterDiePosition[CenterShuttleIndex];

(* Network 219 *)
_e100(CLK := CHoleValve);
_e101(CLK := InCycle);
IF _e100.Q OR _e101.Q THEN ChangeCShuttle := TRUE; END_IF;

(* Network 220 *)
_e102(CLK := Step09);
CShuttleUnlatch := ChangeCShuttle AND _e102.Q;
IF ChangeCShuttle AND _e102.Q THEN ChangeCShuttle := FALSE; END_IF;

(* Network 221 *)
CenterShuttleTemp := ((CenterPosA AND CShuttleUnlatch) OR (CenterShuttleOutput AND NOT CShuttleUnlatch)) AND InCycle;

(* Network 222 *)
CenterShuttleOutput := (CenterShuttleTemp AND NOT InvertShuttle) OR (NOT CenterShuttleTemp AND InvertShuttle AND InCycle);

(* Network 223 *)
RightPosA := RightDiePosition[RightShuttleIndex];

(* Network 224 *)
_e103(CLK := RHoleValve);
_e104(CLK := InCycle);
IF _e103.Q OR _e104.Q THEN ChangeRShuttle := TRUE; END_IF;

(* Network 225 *)
_e105(CLK := Step09);
RShuttleUnlatch := ChangeRShuttle AND _e105.Q;
IF ChangeRShuttle AND _e105.Q THEN ChangeRShuttle := FALSE; END_IF;

(* Network 226 *)
RightShuttleTemp := ((RightPosA AND RShuttleUnlatch) OR (RightShuttleOutput AND NOT RShuttleUnlatch)) AND InCycle;

(* Network 227 *)
RightShuttleOutput := (RightShuttleTemp AND NOT InvertShuttle) OR (NOT RightShuttleTemp AND InvertShuttle AND InCycle);

(* Network 228 *)
UncoilerRunA := InCycle AND NOT InPosition1;
END_PROGRAM
```

#### Variables.var - Local variables
```iecst
VAR
	AnalogForward : BOOL;
	AnalogReverse : BOOL;
	AutoSignal : BOOL;
	BatchCancelUnlatch : BOOL;
	BeadRollFires : BOOL;
	BeadRollUsedUp : BOOL;
	BrakeLatch : BOOL;
	ButtonBack7 : BOOL;
	ButtonFires : BOOL;
	ButtonUsedUp : BOOL;
	CenterHoleFires : BOOL;
	CenterHoleTime : TIME;
	CenterHoleUsedUp : BOOL;
	CenterPosA : BOOL;
	CenterShuttleIndex : INT;
	CenterShuttleTemp : BOOL;
	ChangeCShuttle : BOOL;
	ChangeJob1 : BOOL;
	ChangeLShuttle : BOOL;
	ChangeRShuttle : BOOL;
	CHTemp : BOOL;
	ClearEncoderSignal : BOOL;
	CleatFires : BOOL;
	CleatUsedUp : BOOL;
	CLTTemp : BOOL;
	CShuttleUnlatch : BOOL;
	CustomLTFires : BOOL;
	CustomLTTime : TIME;
	CustomLTUsedUp : BOOL;
	CustomVFires : BOOL;
	CustomVTemp : BOOL;
	CustomVTime : TIME;
	CustomVUsedUp : BOOL;
	DataUpdated : BOOL;
	DDDoneTimer : TON;
	DieDelayDone : BOOL;
	DieUpTime : TIME;
	DirectionDelayDone : BOOL;
	FeedMoveQed : BOOL;
	FinalScan : BOOL;
	GapPulse : BOOL;
	GapTP : BOOL;
	GTime : TIME;
	HalfUpdated1 : BOOL;
	HalfUpdated2 : BOOL;
	IncPartsMade : BOOL;
	InitMoveSignal : BOOL;
	InPositionBand : REAL := 0.01;
	JobChanging : BOOL;
	JobsDifferent : BOOL;
	LeftHoleFires : BOOL;
	LeftHoleTime : TIME;
	LeftHoleUsedUp : BOOL;
	LeftPosA : BOOL;
	LeftShuttleTemp : BOOL;
	LHTemp : BOOL;
	LShuttleUnlatch : BOOL;
	LTFires : BOOL;
	LTTemp : BOOL;
	LTTime : TIME;
	LTUsedUp : BOOL;
	ManualSignal : BOOL;
	MarkAccumulator : REAL;
	MetalEncoderLatch : DINT;
	NewRunJobOk : BOOL;
	NextMoveComplete : BOOL;
	NextMoveLookAgain : BOOL;
	NoShearHits : BOOL;
	PartCutOff : BOOL;
	RHTemp : BOOL;
	RightHoleFires : BOOL;
	RightHoleTime : TIME;
	RightHoleUsedUp : BOOL;
	RightPosA : BOOL;
	RightShuttleTemp : BOOL;
	RShuttleUnlatch : BOOL;
	RTotalInches : REAL;
	RunSpeedCalculated : BOOL;
	SBClampDelay : TIME;
	SBClampDwell : TIME;
	SetConnectorChange : BOOL;
	ShearBrakeFires : BOOL;
	ShearBrakeUsedUp : BOOL;
	ShearFires : BOOL;
	ShearHitsLTZero : BOOL;
	ShearTemp : BOOL;
	shearTime : TIME;
	ShearUsedUp : BOOL;
	SmallResult : REAL;
	SnapButton1 : BOOL;
	SnapButton2 : BOOL;
	SnapButton3 : BOOL;
	SnapButton3A : BOOL;
	SnapButton4 : BOOL;
	SnapButton5 : BOOL;
	SnapButton6 : BOOL;
	Step04A : BOOL;
	Step05A : BOOL;
	Step05B : BOOL;
	Step06 : BOOL;
	Step07 : BOOL;
	Step08 : BOOL;
	Step09 : BOOL;
	Step10 : BOOL;
	Step11 : BOOL;
	Step12 : BOOL;
	Step15 : BOOL;
	Step16 : BOOL;
	Step17 : BOOL;
	Step18 : BOOL;
	Step18A : BOOL;
	Step18B : BOOL;
	Step19 : BOOL;
	ThirdOff1 : BOOL;
	ThirdOff2 : BOOL;
	ThirdOff3 : BOOL;
	TON_0 : TON;
	TON_1 : TON;
	TON_2 : TON;
	TON_3 : TON;
	TON_3Done : BOOL;
	TON_4 : TON;
	TON_4Done : BOOL;
	TON_5 : TON;
	TON_5Done : BOOL;
	TON_6 : TON;
	TON_6Done : BOOL;
	TON_7 : TON;
	TON_7Done : BOOL;
	TON_10 : TON;
	TON_Warning : TON;
	TP_0 : TP;
	TP_1 : TP;
	TP_2 : TP;
	TP_3 : TP;
	TP_4 : TP;
	TP_5 : TP;
	TP_6 : TP;
	TP_7 : TP;
	TP_8 : TP;
	UnlatchBender : BOOL;
	UnlatchButtons : BOOL;
	VFires : BOOL;
	VTemp : BOOL;
	VTime : TIME;
	VUsedUp : BOOL;
	Wait1Ready : BOOL;
	Wait2Ready : BOOL;
	Wait3Ready : BOOL;
	WaitCon1 : BOOL;
	WaitCon2 : BOOL;
	ZCOLT0 : BOOL;
	ZCReverseComplete : BOOL;
	ZCSCTimer : TON;
	ZCSettleComplete : BOOL;
	ZeroCropDifference : DINT;
	ZRCTon : TON;
	TON_8Done : BOOL;
	SnapButton7 : BOOL;
	TON_8 : TON;
END_VAR
```

#### Action.st
```iecst
ACTION myAction:
	(* This was for a test *)
	IF myAction.x AND NOT myAction._x THEN
		FinalScan := TRUE;
	ELSE
	    IF ShearHits < 120000 THEN
			ShearHits := ShearHits + 1;
		END_IF;
	END_IF;

END_ACTION

ACTION getNextMove:
	IF getNextMove.x AND NOT getNextMove._x THEN
		FinalScan := TRUE;
    ELSE
	(*Find smallest move*)
		(*The shear will always be used*)
	NextMoveDone := TRUE;
	SmallResult := ShearMove;
	IF LTNotchMove < SmallResult AND LTNotchMove > InvalidDistREAL THEN
		SmallResult := LTNotchMove;
	END_IF;
	IF VNotchMove < SmallResult AND VNotchMove > InvalidDistREAL THEN
		SmallResult := VNotchMove;
	END_IF;
	IF LeftHoleMove < SmallResult AND LeftHoleMove > InvalidDistREAL THEN
		SmallResult := LeftHoleMove;
	END_IF;
	IF CenterHoleMove < SmallResult AND CenterHoleMove > InvalidDistREAL THEN
		SmallResult := CenterHoleMove;
	END_IF;
	IF RightHoleMove < SmallResult AND RightHoleMove > InvalidDistREAL THEN
		SmallResult := RightHoleMove;
	END_IF;
	IF ButtonMove < SmallResult AND ButtonMove > InvalidDistREAL THEN
		SmallResult := ButtonMove;
	END_IF;
	IF ShearBrakeMove < SmallResult AND ShearBrakeMove > InvalidDistREAL THEN
		SmallResult := ShearBrakeMove;
	END_IF;
	IF CustomLTMove < SmallResult AND CustomLTMove > InvalidDistREAL THEN
		SmallResult := CustomLTMove;
	END_IF;
	IF CleatMove < SmallResult AND CleatMove > InvalidDistREAL THEN
		SmallResult := CleatMove;
	END_IF;
	IF CustomVMove < SmallResult AND CustomVMove > InvalidDistREAL THEN
		SmallResult := CustomVMove;
	END_IF;
	IF BeadRollMove < SmallResult AND BeadRollMove > InvalidDistREAL THEN
		SmallResult := BeadRollMove;
	END_IF;

	ShearMove := ShearMove - SmallResult;
	IF LTNotchMove > InvalidDistREAL THEN
		LTNotchMove := LTNotchMove - SmallResult;
	END_IF;
	IF VNotchMove > InvalidDistREAL THEN
		VNotchMove := VNotchMove - SmallResult;
	END_IF;
	IF LeftHoleMove > InvalidDistREAL THEN
		LeftHoleMove := LeftHoleMove - SmallResult;
	END_IF;
	IF CenterHoleMove > InvalidDistREAL THEN
		CenterHoleMove := CenterHoleMove - SmallResult;
	END_IF;
	IF RightHoleMove > InvalidDistREAL THEN
		RightHoleMove := RightHoleMove - SmallResult;
	END_IF;
	IF ButtonMove > InvalidDistREAL THEN
		ButtonMove := ButtonMove - SmallResult;
	END_IF;
	IF ShearBrakeMove > InvalidDistREAL THEN
		ShearBrakeMove := ShearBrakeMove - SmallResult;
	END_IF;
	IF CustomLTMove > InvalidDistREAL THEN
		CustomLTMove := CustomLTMove - SmallResult;
	END_IF;
	IF CleatMove > InvalidDistREAL THEN
		CleatMove := CleatMove - SmallResult;
	END_IF;
	IF CustomVMove > InvalidDistREAL THEN
		CustomVMove := CustomVMove - SmallResult;
	END_IF;
	IF BeadRollMove > InvalidDistREAL THEN
		BeadRollMove := BeadRollMove - SmallResult;
	END_IF;
  END_IF;
END_ACTION

ACTION UpdateTables:
	IF UpdateTables.x AND NOT UpdateTables._x THEN
		FinalScan := TRUE;
	ELSE
		UpdateTablesDone := TRUE;
		IF ShearUsedUp AND ShearHits > 0 THEN
			ShearFires := TRUE;
			ShearHits := ShearHits - 1;
			(*Do this before the index changes *)
			IF (ShearIndex = 0 AND ShearFFlag = 1) OR
				(ShearIndex = 1 AND ShearTable[2] <= InvalidDistREAL) OR
				(ShearIndex = 2) THEN
				PartCutOff := TRUE;
			END_IF;
				ShearIndex := ShearIndex + 1;
			IF ShearTable[ShearIndex] <= InvalidDistREAL THEN
				ShearIndex := 1;
			END_IF;
			IF ShearHits <= 0 THEN
				MakeShearTable := TRUE;
				ShearIndex := 0;
			END_IF;
		END_IF;
		IF LTUsedUp THEN
			IF LTNotchHits > 0 THEN
				LTFires := TRUE;
				LTNotchHits := LTNotchHits - 1;
			END_IF;
			LTNotchIndex := LTNotchIndex + 1;
			IF LTNotchTable[LTNotchIndex] <= InvalidDistREAL THEN
				LTNotchIndex := 1;
			END_IF;
			SavedConnector := LatestConnector;
			IF LTNotchHits <= 0 THEN
				MakeLTTable := TRUE;
				LTNotchIndex := 0;
			END_IF;
		END_IF;
		IF VUsedUp THEN
			IF VNotchHits > 0 THEN
				VFires := TRUE;
				VNotchHits := VNotchHits - 1;
			END_IF;
			VNotchIndex := VNotchIndex + 1;
			IF VNotchTable[VNotchIndex] <= InvalidDistREAL THEN
				VNotchIndex := 1;
			END_IF;
			IF VNotchHits <= 0 THEN
				MakeVTable := TRUE;
				VNotchIndex := 0;
			END_IF;
		END_IF;
		IF LeftHoleUsedUp THEN
			IF LeftHoleHits > 0 THEN
				LeftHoleFires := TRUE;
				LeftHoleHits := LeftHoleHits - 1;
			END_IF;
			LeftHoleIndex := LeftHoleIndex + 1;
			IF LeftHoleTable[LeftHoleIndex] <= InvalidDistREAL THEN
				LeftHoleIndex := 1;
			END_IF;
			IF LeftHoleHits <= 0 THEN
				MakeLHoleTable := TRUE;
				LeftHoleIndex := 0;
			END_IF;
		END_IF;
		IF CenterHoleUsedUp THEN
			IF CenterHoleHits > 0 THEN
				CenterHoleFires := TRUE;
				CenterHoleHits := CenterHoleHits - 1;
			END_IF;
			CenterHoleIndex := CenterHoleIndex + 1;
			IF CenterHoleTable[CenterHoleIndex] <= InvalidDistREAL THEN
				CenterHoleIndex := 1;
			END_IF;
			IF CenterHoleHits <= 0 THEN
				MakeCHoleTable := TRUE;
				CenterHoleIndex := 0;
			END_IF;
		END_IF;
		IF RightHoleUsedUp THEN
			IF RightHoleHits > 0 THEN
				RightHoleFires := TRUE;
				RightHoleHits := RightHoleHits - 1;
			END_IF;
			RightHoleIndex := RightHoleIndex + 1;
			IF RightHoleTable[RightHoleIndex] <= InvalidDistREAL THEN
				RightHoleIndex := 1;
			END_IF;
			IF RightHoleHits <= 0 THEN
				MakeRHoleTable := TRUE;
				RightHoleIndex := 0;
			END_IF;
		END_IF
		IF ButtonUsedUp THEN
			IF ButtonHits > 0 THEN
				ButtonFires := TRUE;
				ButtonHits := ButtonHits - 1;
			END_IF;
			ButtonIndex := ButtonIndex + 1;
			IF ButtonTable[ButtonIndex] <= InvalidDistREAL THEN
				ButtonIndex := 1;
			END_IF;
			IF ButtonHits <= 0 THEN
				MakeButtonTable := TRUE;
				ButtonIndex := 0;
			END_IF;
		END_IF;
		IF ShearBrakeUsedUp THEN
			IF ShearBrakeHits > 0 THEN
				ShearBrakeFires := TRUE;
				ShearBrakeHits := ShearBrakeHits - 1;
			END_IF;
			ShearBrakeIndex := ShearBrakeIndex + 1;
			IF ShearBrakeTable[ShearBrakeIndex] <= InvalidDistREAL THEN
				ShearBrakeIndex := 1;
			END_IF;
			IF ShearBrakeHits <= 0 THEN
				MakeShearBrakeTable := TRUE;
				ShearBrakeIndex := 0;
			END_IF;
		END_IF;
		IF CustomLTUsedUp THEN
			IF CustomLTHits > 0 THEN
				CustomLTFires := TRUE;
				CustomLTHits := CustomLTHits - 1;
			END_IF;
			CustomLTIndex := CustomLTIndex + 1;
			IF CustomLTTable[CustomLTIndex] <= InvalidDistREAL THEN
				CustomLTIndex := 1;
			END_IF;
			IF CustomLTHits <= 0 THEN
				MakeCustomLTTable := TRUE;
				CustomLTIndex := 0;
			END_IF;
		END_IF;
		IF CleatUsedUp THEN
			IF CleatHits > 0 THEN
				CleatFires := TRUE;
				CleatHits := CleatHits - 1;
			END_IF;
			CleatIndex := CleatIndex + 1;
			IF CleatTable[CleatIndex] <= InvalidDistREAL THEN
				CleatIndex := 1;
			END_IF;
			IF CleatHits <= 0 THEN
				MakeCleatTable := TRUE;
				CleatIndex := 0;
			END_IF;
		END_IF;
		IF CustomVUsedUp THEN
			IF CustomVHits > 0 THEN
				CustomVFires := TRUE;
				CustomVHits := CustomVHits - 1;
			END_IF;
			CustomVIndex := CustomVIndex + 1;
			IF CustomVTable[CustomVIndex] <= InvalidDistREAL THEN
				CustomVIndex := 1;
			END_IF;
			IF CustomVHits <= 0 THEN
				MakeCustomVTable := TRUE;
				CustomVIndex := 0;
			END_IF;
		END_IF;
		IF BeadRollUsedUp THEN
			IF BeadRollHits > 0 THEN
				BeadRollFires := TRUE;
				BeadRollHits := BeadRollHits - 1;
			END_IF;
			BeadRollIndex := BeadRollIndex + 1;
			IF BeadRollTable[BeadRollIndex] <= InvalidDistREAL THEN
				BeadRollIndex := 1;
			END_IF;
			IF BeadRollHits <= 0 THEN
				MakeBeadRollTable := TRUE;
				BeadRollIndex := 0;
			END_IF;
	    END_IF;
	END_IF;
END_ACTION
```

### Program Logical/HMIButtons (IEC)

#### Variables.var
```iecst
VAR
	BlockingValveUnlatch : BOOL;
	ZeroCropUnlatch : BOOL;
	ZeroCropSignal : BOOL;
END_VAR
```

#### Cyclic.ld
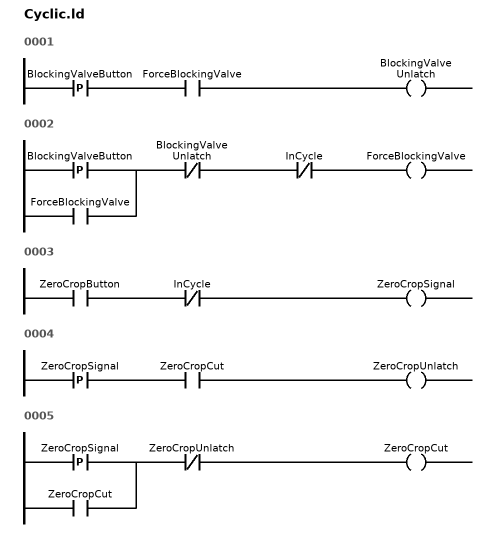
Ladder, written as Structured Text:
```iecst
PROGRAM _CYCLIC
VAR
    _e1 : R_TRIG;
    _e2 : R_TRIG;
    _e3 : R_TRIG;
    _e4 : R_TRIG;
END_VAR
(* Network 1 *)
_e1(CLK := BlockingValveButton);
BlockingValveUnlatch := _e1.Q AND ForceBlockingValve;

(* Network 2 *)
_e2(CLK := BlockingValveButton);
ForceBlockingValve := (_e2.Q OR ForceBlockingValve) AND NOT BlockingValveUnlatch AND NOT InCycle;

(* Network 3 *)
ZeroCropSignal := ZeroCropButton AND NOT InCycle;

(* Network 4 *)
_e3(CLK := ZeroCropSignal);
ZeroCropUnlatch := _e3.Q AND ZeroCropCut;

(* Network 5 *)
_e4(CLK := ZeroCropSignal);
ZeroCropCut := (_e4.Q OR ZeroCropCut) AND NOT ZeroCropUnlatch;
END_PROGRAM
```

- OpcTag.opct (not shown)

### LibAsTCP1_ST.typ - Global Datatype
```iecst
(********************************************************************
 * COPYRIGHT -- Bernecker + Rainer
 ********************************************************************
 * Package: LibAsTCP
 * File: LibAsTCP.typ
 * Author: Bernecker + Rainer
 * Created: February 21, 2008
 ********************************************************************
 * Data types of package LibAsTCP
 ********************************************************************)

TYPE
	LibAsTCP1_ST_typ : 	STRUCT  (*Datatyp for global Variables*)
		receive_data : ARRAY[0..100]OF UDINT; (*Data which has been received*)
		send_data : ARRAY[0..100]OF BYTE; (*Data which should be sent*)
	END_STRUCT;
END_TYPE
```

### Program Logical/LibAsTCP1_ST/Server (IEC) - AsTCP Server Application
